PROGRAM UR5_robot
VAR
//banderas



i : BOOL := FALSE;
i2 : BOOL := FALSE;

vi_get_img : BOOL;
vi_img_ok: BOOL;

cx : REAL;
cy : REAL;
giro : REAL;
centro_ok : BOOL;
motor_pos_ok : BOOL;


// variables cabezal
giro_cabezal_dere : REAL;

vi_img_cabezal_dere_ok : BOOL;
vi_img_cabezal_dere_proc_ok : BOOL;
vi_get_img_cabezal_dere : BOOL;
vi_get_img_tuerca : BOOL;
giro_desartonillado : REAL;
cal_vueltas : REAL;
giro_aux_int : DINT;
giro_aux_float : REAL;

Atornillar: INT;
END_VAR

VAR_INPUT	
iniciar: BOOL := FALSE;
END_VAR

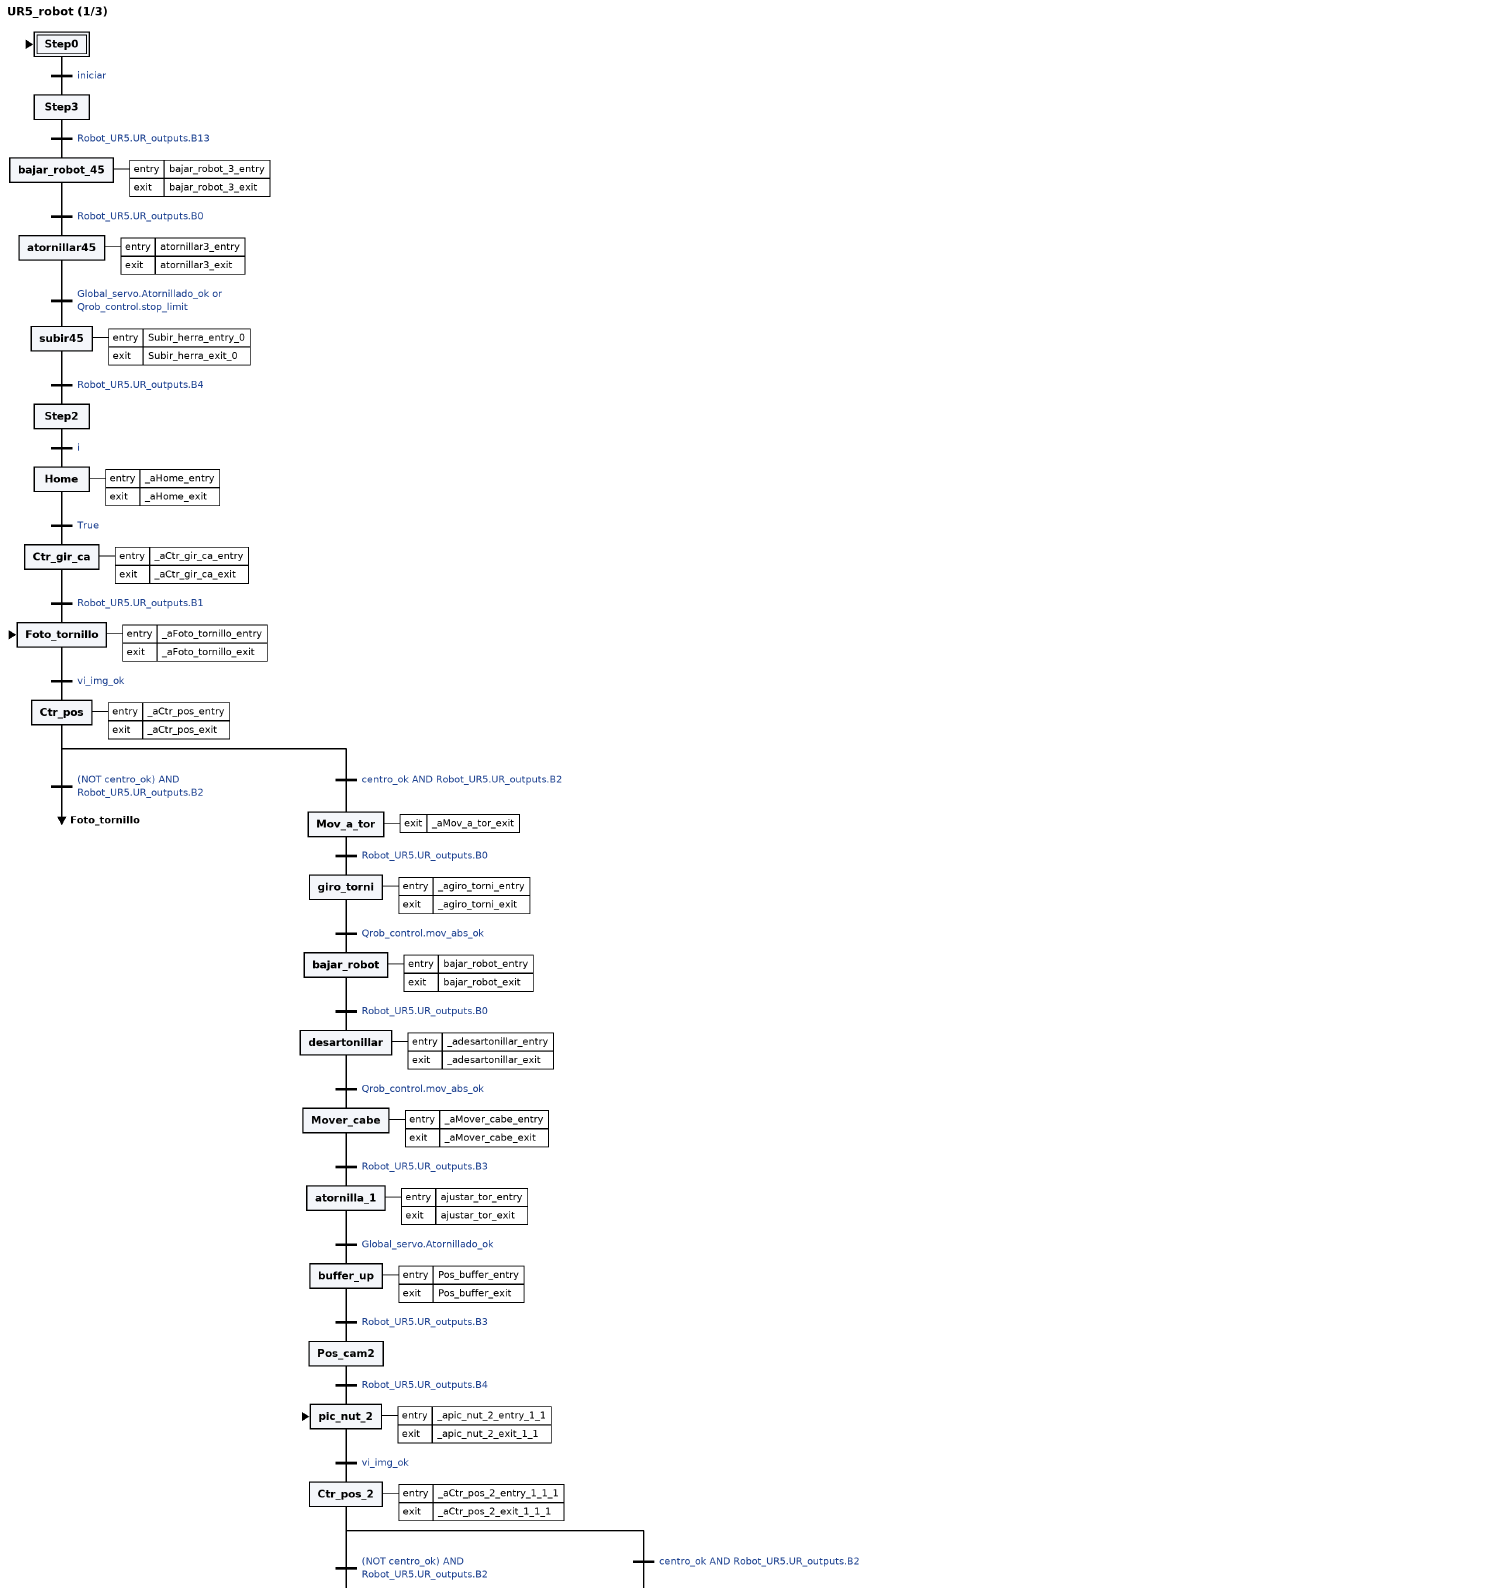
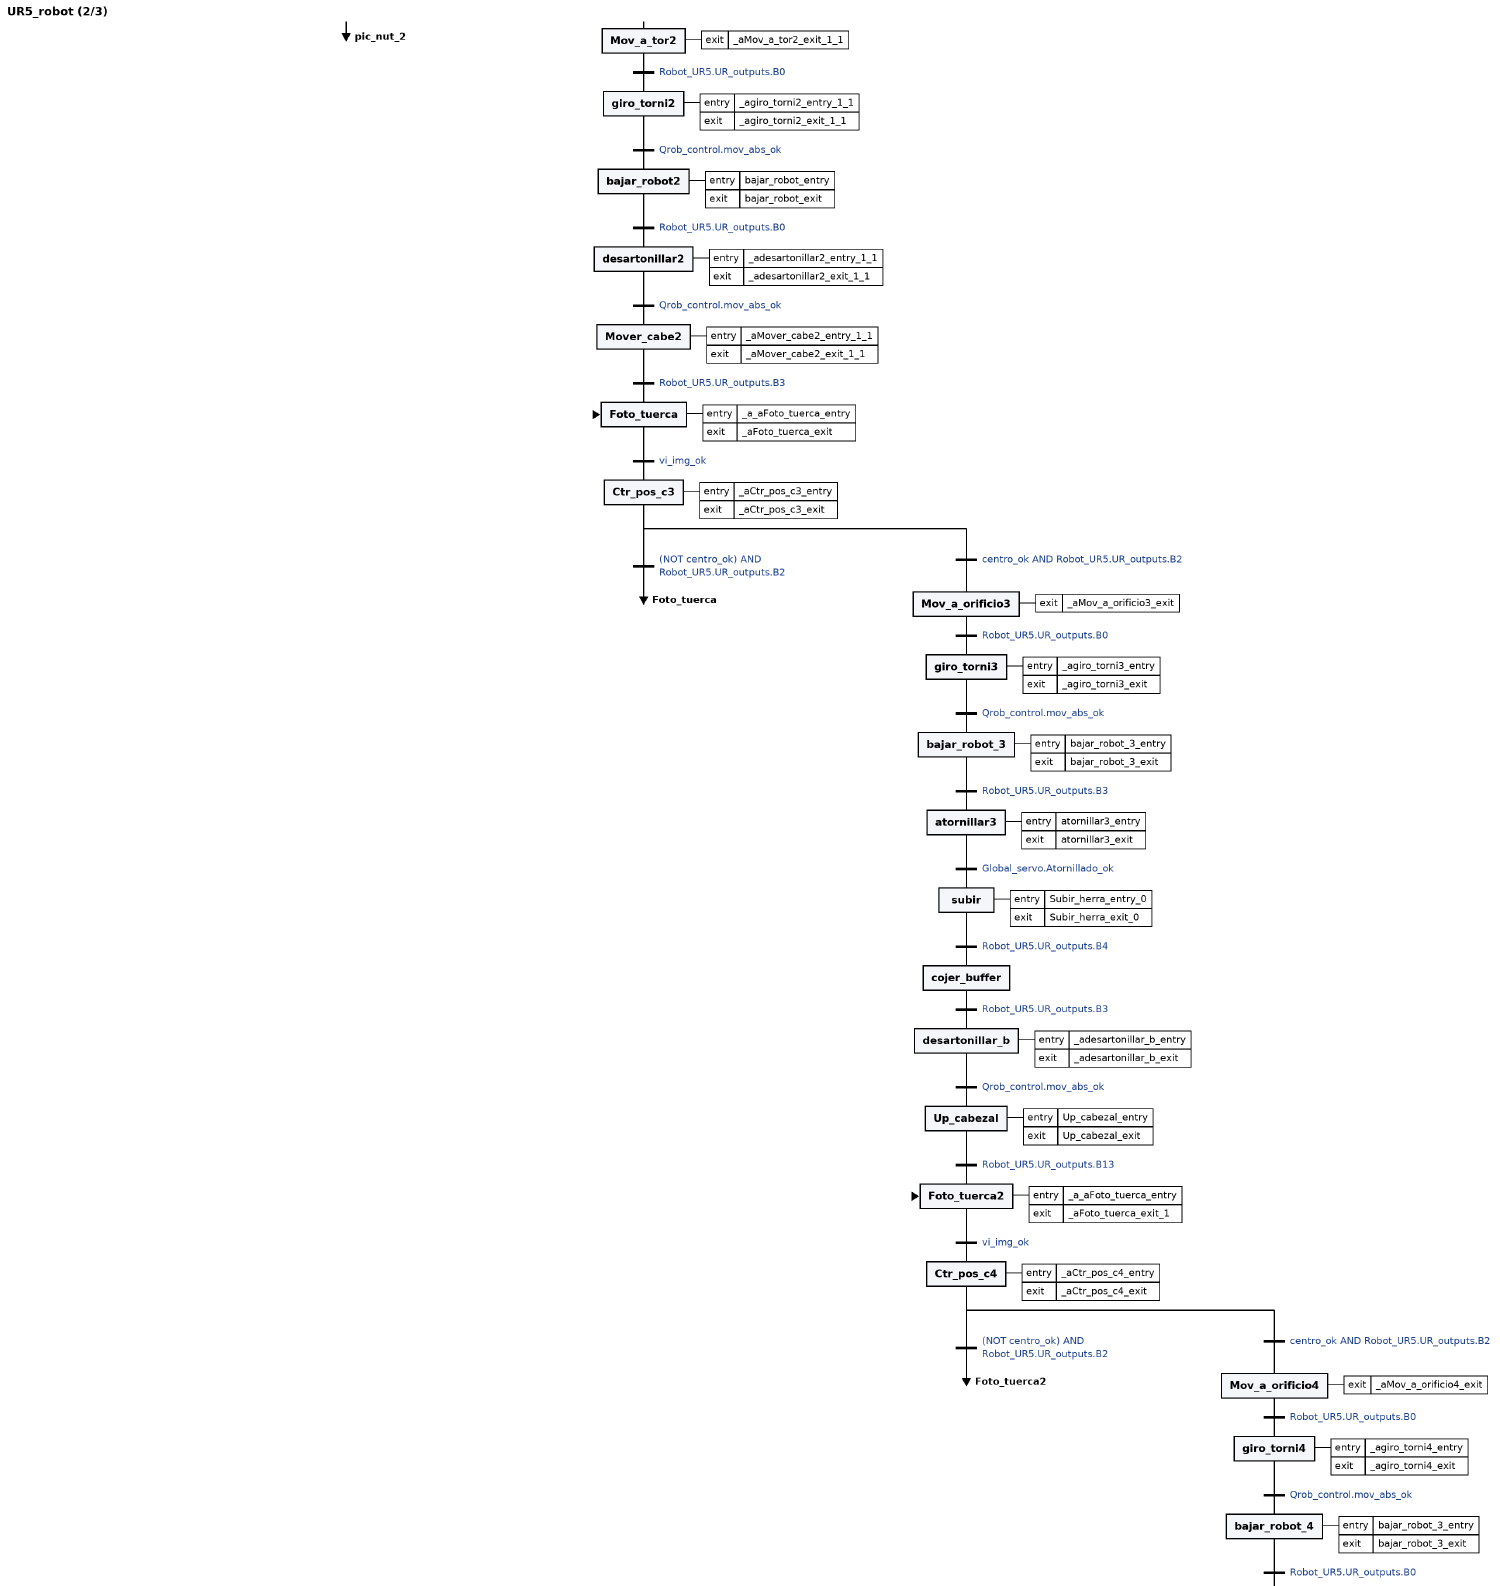
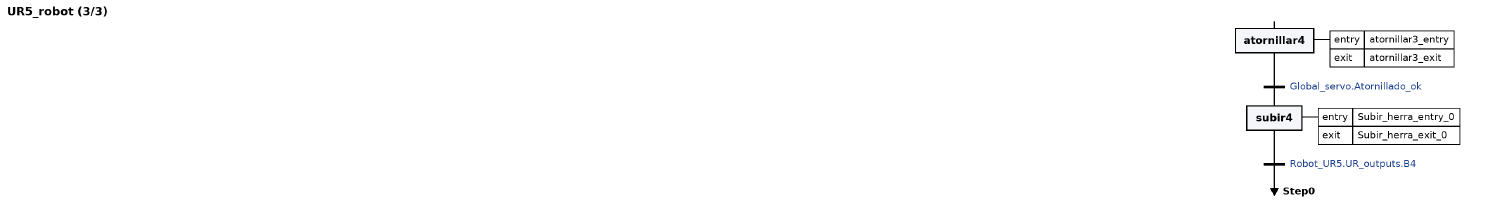
INITIAL_STEP Step0:
END_STEP
TRANSITION FROM Step0 TO Step3
    := iniciar;
END_TRANSITION
// macro Macro0 begins
STEP Step3:
END_STEP
TRANSITION FROM Step3 TO bajar_robot_45
    := Robot_UR5.UR_outputs.B13;
END_TRANSITION
STEP bajar_robot_45:
    bajar_robot_3_entry(P1);  // entry action
    bajar_robot_3_exit(P0);  // exit action
END_STEP
TRANSITION FROM bajar_robot_45 TO atornillar45
    := Robot_UR5.UR_outputs.B0;
END_TRANSITION
STEP atornillar45:
    atornillar3_entry(P1);  // entry action
    atornillar3_exit(P0);  // exit action
END_STEP
TRANSITION FROM atornillar45 TO subir45
    := Global_servo.Atornillado_ok or Qrob_control.stop_limit;
END_TRANSITION
STEP subir45:
    Subir_herra_entry_0(P1);  // entry action
    Subir_herra_exit_0(P0);  // exit action
END_STEP
TRANSITION FROM subir45 TO Step2
    := Robot_UR5.UR_outputs.B4;
END_TRANSITION
STEP Step2:
END_STEP
TRANSITION FROM Step2 TO Home
    := i;
END_TRANSITION
STEP Home:
    _aHome_entry(P1);  // entry action
    _aHome_exit(P0);  // exit action
END_STEP
TRANSITION FROM Home TO Ctr_gir_ca
    := True;
END_TRANSITION
STEP Ctr_gir_ca:
    _aCtr_gir_ca_entry(P1);  // entry action
    _aCtr_gir_ca_exit(P0);  // exit action
END_STEP
TRANSITION FROM Ctr_gir_ca TO Foto_tornillo
    := Robot_UR5.UR_outputs.B1;
END_TRANSITION
STEP Foto_tornillo:
    _aFoto_tornillo_entry(P1);  // entry action
    _aFoto_tornillo_exit(P0);  // exit action
END_STEP
TRANSITION FROM Foto_tornillo TO Ctr_pos
    := vi_img_ok;
END_TRANSITION
STEP Ctr_pos:
    _aCtr_pos_entry(P1);  // entry action
    _aCtr_pos_exit(P0);  // exit action
END_STEP
TRANSITION FROM Ctr_pos TO Foto_tornillo
    := (NOT centro_ok) AND Robot_UR5.UR_outputs.B2;
END_TRANSITION
TRANSITION FROM Ctr_pos TO Mov_a_tor
    := centro_ok AND Robot_UR5.UR_outputs.B2;
END_TRANSITION
STEP Mov_a_tor:
    _aMov_a_tor_exit(P0);  // exit action
END_STEP
TRANSITION FROM Mov_a_tor TO giro_torni
    := Robot_UR5.UR_outputs.B0;
END_TRANSITION
STEP giro_torni:
    _agiro_torni_entry(P1);  // entry action
    _agiro_torni_exit(P0);  // exit action
END_STEP
TRANSITION FROM giro_torni TO bajar_robot
    := Qrob_control.mov_abs_ok;
END_TRANSITION
STEP bajar_robot:
    bajar_robot_entry(P1);  // entry action
    bajar_robot_exit(P0);  // exit action
END_STEP
TRANSITION FROM bajar_robot TO desartonillar
    := Robot_UR5.UR_outputs.B0;
END_TRANSITION
STEP desartonillar:
    _adesartonillar_entry(P1);  // entry action
    _adesartonillar_exit(P0);  // exit action
END_STEP
TRANSITION FROM desartonillar TO Mover_cabe
    := Qrob_control.mov_abs_ok;
END_TRANSITION
STEP Mover_cabe:
    _aMover_cabe_entry(P1);  // entry action
    _aMover_cabe_exit(P0);  // exit action
END_STEP
TRANSITION FROM Mover_cabe TO atornilla_1
    := Robot_UR5.UR_outputs.B3;
END_TRANSITION
STEP atornilla_1:
    ajustar_tor_entry(P1);  // entry action
    ajustar_tor_exit(P0);  // exit action
END_STEP
TRANSITION FROM atornilla_1 TO buffer_up
    := Global_servo.Atornillado_ok;
END_TRANSITION
STEP buffer_up:
    Pos_buffer_entry(P1);  // entry action
    Pos_buffer_exit(P0);  // exit action
END_STEP
TRANSITION FROM buffer_up TO Pos_cam2
    := Robot_UR5.UR_outputs.B3;
END_TRANSITION
STEP Pos_cam2:
END_STEP
TRANSITION FROM Pos_cam2 TO pic_nut_2
    := Robot_UR5.UR_outputs.B4;
END_TRANSITION
STEP pic_nut_2:
    _apic_nut_2_entry_1_1(P1);  // entry action
    _apic_nut_2_exit_1_1(P0);  // exit action
END_STEP
TRANSITION FROM pic_nut_2 TO Ctr_pos_2
    := vi_img_ok;
END_TRANSITION
STEP Ctr_pos_2:
    _aCtr_pos_2_entry_1_1_1(P1);  // entry action
    _aCtr_pos_2_exit_1_1_1(P0);  // exit action
END_STEP
TRANSITION FROM Ctr_pos_2 TO pic_nut_2
    := (NOT centro_ok) AND Robot_UR5.UR_outputs.B2;
END_TRANSITION
TRANSITION FROM Ctr_pos_2 TO Mov_a_tor2
    := centro_ok AND Robot_UR5.UR_outputs.B2;
END_TRANSITION
STEP Mov_a_tor2:
    _aMov_a_tor2_exit_1_1(P0);  // exit action
END_STEP
TRANSITION FROM Mov_a_tor2 TO giro_torni2
    := Robot_UR5.UR_outputs.B0;
END_TRANSITION
STEP giro_torni2:
    _agiro_torni2_entry_1_1(P1);  // entry action
    _agiro_torni2_exit_1_1(P0);  // exit action
END_STEP
TRANSITION FROM giro_torni2 TO bajar_robot2
    := Qrob_control.mov_abs_ok;
END_TRANSITION
STEP bajar_robot2:
    bajar_robot_entry(P1);  // entry action
    bajar_robot_exit(P0);  // exit action
END_STEP
TRANSITION FROM bajar_robot2 TO desartonillar2
    := Robot_UR5.UR_outputs.B0;
END_TRANSITION
STEP desartonillar2:
    _adesartonillar2_entry_1_1(P1);  // entry action
    _adesartonillar2_exit_1_1(P0);  // exit action
END_STEP
TRANSITION FROM desartonillar2 TO Mover_cabe2
    := Qrob_control.mov_abs_ok;
END_TRANSITION
STEP Mover_cabe2:
    _aMover_cabe2_entry_1_1(P1);  // entry action
    _aMover_cabe2_exit_1_1(P0);  // exit action
END_STEP
TRANSITION FROM Mover_cabe2 TO Foto_tuerca
    := Robot_UR5.UR_outputs.B3;
END_TRANSITION
STEP Foto_tuerca:
    _a_aFoto_tuerca_entry(P1);  // entry action
    _aFoto_tuerca_exit(P0);  // exit action
END_STEP
TRANSITION FROM Foto_tuerca TO Ctr_pos_c3
    := vi_img_ok;
END_TRANSITION
STEP Ctr_pos_c3:
    _aCtr_pos_c3_entry(P1);  // entry action
    _aCtr_pos_c3_exit(P0);  // exit action
END_STEP
TRANSITION FROM Ctr_pos_c3 TO Foto_tuerca
    := (NOT centro_ok) AND Robot_UR5.UR_outputs.B2;
END_TRANSITION
TRANSITION FROM Ctr_pos_c3 TO Mov_a_orificio3
    := centro_ok AND Robot_UR5.UR_outputs.B2;
END_TRANSITION
STEP Mov_a_orificio3:
    _aMov_a_orificio3_exit(P0);  // exit action
END_STEP
TRANSITION FROM Mov_a_orificio3 TO giro_torni3
    := Robot_UR5.UR_outputs.B0;
END_TRANSITION
STEP giro_torni3:
    _agiro_torni3_entry(P1);  // entry action
    _agiro_torni3_exit(P0);  // exit action
END_STEP
TRANSITION FROM giro_torni3 TO bajar_robot_3
    := Qrob_control.mov_abs_ok;
END_TRANSITION
STEP bajar_robot_3:
    bajar_robot_3_entry(P1);  // entry action
    bajar_robot_3_exit(P0);  // exit action
END_STEP
TRANSITION FROM bajar_robot_3 TO atornillar3
    := Robot_UR5.UR_outputs.B3;
END_TRANSITION
STEP atornillar3:
    atornillar3_entry(P1);  // entry action
    atornillar3_exit(P0);  // exit action
END_STEP
TRANSITION FROM atornillar3 TO subir
    := Global_servo.Atornillado_ok;
END_TRANSITION
STEP subir:
    Subir_herra_entry_0(P1);  // entry action
    Subir_herra_exit_0(P0);  // exit action
END_STEP
TRANSITION FROM subir TO cojer_buffer
    := Robot_UR5.UR_outputs.B4;
END_TRANSITION
STEP cojer_buffer:
END_STEP
TRANSITION FROM cojer_buffer TO desartonillar_b
    := Robot_UR5.UR_outputs.B3;
END_TRANSITION
STEP desartonillar_b:
    _adesartonillar_b_entry(P1);  // entry action
    _adesartonillar_b_exit(P0);  // exit action
END_STEP
TRANSITION FROM desartonillar_b TO Up_cabezal
    := Qrob_control.mov_abs_ok;
END_TRANSITION
STEP Up_cabezal:
    Up_cabezal_entry(P1);  // entry action
    Up_cabezal_exit(P0);  // exit action
END_STEP
TRANSITION FROM Up_cabezal TO Foto_tuerca2
    := Robot_UR5.UR_outputs.B13;
END_TRANSITION
STEP Foto_tuerca2:
    _a_aFoto_tuerca_entry(P1);  // entry action
    _aFoto_tuerca_exit_1(P0);  // exit action
END_STEP
TRANSITION FROM Foto_tuerca2 TO Ctr_pos_c4
    := vi_img_ok;
END_TRANSITION
STEP Ctr_pos_c4:
    _aCtr_pos_c4_entry(P1);  // entry action
    _aCtr_pos_c4_exit(P0);  // exit action
END_STEP
TRANSITION FROM Ctr_pos_c4 TO Foto_tuerca2
    := (NOT centro_ok) AND Robot_UR5.UR_outputs.B2;
END_TRANSITION
TRANSITION FROM Ctr_pos_c4 TO Mov_a_orificio4
    := centro_ok AND Robot_UR5.UR_outputs.B2;
END_TRANSITION
STEP Mov_a_orificio4:
    _aMov_a_orificio4_exit(P0);  // exit action
END_STEP
TRANSITION FROM Mov_a_orificio4 TO giro_torni4
    := Robot_UR5.UR_outputs.B0;
END_TRANSITION
STEP giro_torni4:
    _agiro_torni4_entry(P1);  // entry action
    _agiro_torni4_exit(P0);  // exit action
END_STEP
TRANSITION FROM giro_torni4 TO bajar_robot_4
    := Qrob_control.mov_abs_ok;
END_TRANSITION
STEP bajar_robot_4:
    bajar_robot_3_entry(P1);  // entry action
    bajar_robot_3_exit(P0);  // exit action
END_STEP
TRANSITION FROM bajar_robot_4 TO atornillar4
    := Robot_UR5.UR_outputs.B0;
END_TRANSITION
STEP atornillar4:
    atornillar3_entry(P1);  // entry action
    atornillar3_exit(P0);  // exit action
END_STEP
TRANSITION FROM atornillar4 TO subir4
    := Global_servo.Atornillado_ok;
END_TRANSITION
STEP subir4:
    Subir_herra_entry_0(P1);  // entry action
    Subir_herra_exit_0(P0);  // exit action
END_STEP
TRANSITION FROM subir4 TO Step0
    := Robot_UR5.UR_outputs.B4;
END_TRANSITION

ACTION _a_aFoto_tuerca_entry:


vi_get_img_tuerca := True;
END_ACTION

ACTION _aCtr_gir_ca_entry:
Robot_UR5.UR_inputs.Floats.FLOAT3 := flip_real(data_to_robot.head_roll_right);
Robot_UR5.UR_inputs.Floats.FLOAT4 := flip_real(data_to_robot.head_roll_left);
Robot_UR5.UR_inputs.Bits.B0 := TRUE;
END_ACTION

ACTION _aCtr_gir_ca_exit:
Robot_UR5.UR_inputs.Bits.B0 := False;
END_ACTION

ACTION _aCtr_pos_2_entry_1_1_1:
vi_img_ok := FALSE;

Robot_UR5.UR_inputs.Floats.FLOAT0 := flip_real(cx);
Robot_UR5.UR_inputs.Floats.FLOAT1 := flip_real(cy);
Robot_UR5.UR_inputs.Floats.FLOAT2 := flip_real(giro);


IF ( ABS(cx) < 1) AND ( ABS(cy) < 1) THEN 
Robot_UR5.UR_inputs.Bits.B3 := TRUE;
centro_ok := TRUE;
ELSE 
Robot_UR5.UR_inputs.Bits.B3 := FALSE;
centro_ok := FALSE;	
END_IF

Robot_UR5.UR_inputs.Bits.B2 := TRUE;
END_ACTION

ACTION _aCtr_pos_2_exit_1_1_1:
Robot_UR5.UR_inputs.Bits.B2 := False;
END_ACTION

ACTION _aCtr_pos_c3_entry:
vi_img_ok := FALSE;

Robot_UR5.UR_inputs.Floats.FLOAT0 := flip_real(cx);
Robot_UR5.UR_inputs.Floats.FLOAT1 := flip_real(cy);



IF ( ABS(cx) < 0.5) AND ( ABS(cy) < 0.5) THEN 
Robot_UR5.UR_inputs.Bits.B3 := TRUE;
centro_ok := TRUE;
ELSE 
Robot_UR5.UR_inputs.Bits.B3 := FALSE;
centro_ok := FALSE;	
END_IF

Robot_UR5.UR_inputs.Bits.B2 := TRUE;
END_ACTION

ACTION _aCtr_pos_c3_exit:
Robot_UR5.UR_inputs.Bits.B2 := False;
END_ACTION

ACTION _aCtr_pos_c4_entry:
vi_img_ok := FALSE;

Robot_UR5.UR_inputs.Floats.FLOAT0 := flip_real(cx);
Robot_UR5.UR_inputs.Floats.FLOAT1 := flip_real(cy);



IF ( ABS(cx) < 0.5) AND ( ABS(cy) < 0.5) THEN 
Robot_UR5.UR_inputs.Bits.B3 := TRUE;
centro_ok := TRUE;
ELSE 
Robot_UR5.UR_inputs.Bits.B3 := FALSE;
centro_ok := FALSE;	
END_IF

Robot_UR5.UR_inputs.Bits.B2 := TRUE;
END_ACTION

ACTION _aCtr_pos_c4_exit:
Robot_UR5.UR_inputs.Bits.B2 := False;
END_ACTION

ACTION _aCtr_pos_entry:
vi_img_ok := FALSE;

Robot_UR5.UR_inputs.Floats.FLOAT0 := flip_real(cx);
Robot_UR5.UR_inputs.Floats.FLOAT1 := flip_real(cy);
Robot_UR5.UR_inputs.Floats.FLOAT2 := flip_real(giro);


IF ( ABS(cx) < 1) AND ( ABS(cy) < 1) THEN 
Robot_UR5.UR_inputs.Bits.B3 := TRUE;
centro_ok := TRUE;
ELSE 
Robot_UR5.UR_inputs.Bits.B3 := FALSE;
centro_ok := FALSE;	
END_IF

Robot_UR5.UR_inputs.Bits.B2 := TRUE;
END_ACTION

ACTION _aCtr_pos_exit:
Robot_UR5.UR_inputs.Bits.B2 := False;
END_ACTION

ACTION _adesartonillar_b_entry:




giro_desartonillado :=  (-24*360) + Qrob_control.actual_position;
Qrob_control.pos_mover_abs := giro_desartonillado;
Qrob_control.velocidad := 150;


Qrob_control.mover_abs := TRUE;
END_ACTION

ACTION _adesartonillar_b_exit:
Qrob_control.mover_abs := FALSE;
END_ACTION

ACTION _adesartonillar_entry:




giro_desartonillado := giro -(15*360);
//giro_desartonillado := giro -2160;
Qrob_control.pos_mover_abs := giro_desartonillado;
Qrob_control.velocidad := 150;


Qrob_control.mover_abs := TRUE;
END_ACTION

ACTION _adesartonillar_exit:
Qrob_control.mover_abs := FALSE;
END_ACTION

ACTION _adesartonillar2_entry_1_1:





giro_desartonillado := giro -(15*360);
//giro_desartonillado := giro -2160;
Qrob_control.pos_mover_abs := giro_desartonillado;
Qrob_control.velocidad := 150;


Qrob_control.mover_abs := TRUE;
END_ACTION

ACTION _adesartonillar2_exit_1_1:
Qrob_control.mover_abs := FALSE;
END_ACTION

ACTION _aFoto_tornillo_entry:
vi_get_img := True;
END_ACTION

ACTION _aFoto_tornillo_entry_1:
vi_get_img := True;
END_ACTION

ACTION _aFoto_tornillo_exit:
vi_get_img := False;
END_ACTION

ACTION _aFoto_tuerca_exit:

vi_get_img_tuerca := False;
END_ACTION

ACTION _aFoto_tuerca_exit_1:

vi_get_img_tuerca := False;
END_ACTION

ACTION _agiro_torni_entry:
//POU.detener := TRUE;
//Pou.detener := FALSE;


//home qrob while angle
giro_aux_int := ABS(TRUNC(Qrob_control.actual_position/360));
giro_aux_float := ABS( - (Qrob_control.actual_position/360));
giro_aux_float := -1*(giro_aux_float*360);






Qrob_control.velocidad := 50;
//Qrob_control.pos_mover_abs := giro;
Qrob_control.pos_mover_abs := (Qrob_control.actual_position + giro_aux_float) + giro;
Qrob_control.mover_abs := TRUE;
END_ACTION

ACTION _agiro_torni_exit:
Qrob_control.mover_abs := FALSE;
END_ACTION

ACTION _agiro_torni2_entry_1_1:
//POU.detener := TRUE;
//Pou.detener := FALSE;


//home qrob while angle
giro_aux_int := ABS(TRUNC(Qrob_control.actual_position/360));
giro_aux_float := ABS(giro_aux_int- (Qrob_control.actual_position/360));
giro_aux_float := -1*(giro_aux_float*360);






Qrob_control.velocidad := 50;
//Qrob_control.pos_mover_abs := giro;
Qrob_control.pos_mover_abs := (Qrob_control.actual_position + giro_aux_float) + giro;
giro := Qrob_control.pos_mover_abs;
Qrob_control.mover_abs := TRUE;
END_ACTION

ACTION _agiro_torni2_exit_1_1:
Qrob_control.mover_abs := FALSE;
END_ACTION

ACTION _agiro_torni3_entry:
//POU.detener := TRUE;
//Pou.detener := FALSE;


giro_aux_int := TRUNC(Qrob_control.actual_position/360);

giro_aux_float := ABS(giro_aux_int- (Qrob_control.actual_position/360));
giro_aux_float := -1*(giro_aux_float*360);

Qrob_control.velocidad := 100;
Qrob_control.pos_mover_abs := Qrob_control.actual_position + giro_aux_float;
Qrob_control.mover_abs := TRUE;
END_ACTION

ACTION _agiro_torni3_exit:
Qrob_control.mover_abs := FALSE;
END_ACTION

ACTION _agiro_torni4_entry:
//POU.detener := TRUE;
//Pou.detener := FALSE;

//Qrob_control.velocidad := 100;
//Qrob_control.pos_mover_abs := 0;
//Qrob_control.mover_abs := TRUE;


giro_aux_int := TRUNC(Qrob_control.actual_position/360);

giro_aux_float := ABS(giro_aux_int- (Qrob_control.actual_position/360));
giro_aux_float := -1*(giro_aux_float*360);

Qrob_control.velocidad := 100;
Qrob_control.pos_mover_abs := Qrob_control.actual_position + giro_aux_float;
Qrob_control.mover_abs := TRUE;
END_ACTION

ACTION _agiro_torni4_exit:
Qrob_control.mover_abs := FALSE;
END_ACTION

ACTION _aHome_entry:
i := FALSE;
Robot_UR5.UR_inputs.Bits.B0 := TRUE;
//POU.EnableAxis1 := True;
giro :=0;
//Qrob_control.ajustar_tornillo := FALSE;
//Qrob_control.pos_mover_abs := 0;
//Qrob_control.velocidad := 100;


//Qrob_control.mover_abs := TRUE;
END_ACTION

ACTION _aHome_exit:
Robot_UR5.UR_inputs.Bits.B0 := FALSE;
iniciar := FALSE;
Qrob_control.mover_abs := False;
END_ACTION

ACTION _aMov_a_orificio3_exit:
Robot_UR5.UR_inputs.Bits.B2 := FALSE;
END_ACTION

ACTION _aMov_a_orificio4_exit:
Robot_UR5.UR_inputs.Bits.B2 := FALSE;
END_ACTION

ACTION _aMov_a_tor_exit:
Robot_UR5.UR_inputs.Bits.B2 := FALSE;
END_ACTION

ACTION _aMov_a_tor2_exit_1_1:
Robot_UR5.UR_inputs.Bits.B2 := FALSE;
END_ACTION

ACTION _aMover_cabe_entry:
Robot_UR5.UR_inputs.Bits.B5 := True;
END_ACTION

ACTION _aMover_cabe_exit:
Robot_UR5.UR_inputs.Bits.B5 := False;
END_ACTION

ACTION _aMover_cabe2_entry_1_1:
Robot_UR5.UR_inputs.Bits.B5 := True;
END_ACTION

ACTION _aMover_cabe2_exit_1_1:
Robot_UR5.UR_inputs.Bits.B5 := False;
END_ACTION

ACTION _apic_nut_2_entry_1_1:
vi_get_img := True;
END_ACTION

ACTION _apic_nut_2_exit_1_1:
vi_get_img := False;
END_ACTION

ACTION ajustar_tor_entry:


//Atornillado_funcion(Iniciar:= TRUE, Corriente := 60, vueltas := 8, giro_alivio := 3);

Atornillar_CS.UR5.Corriente := 10;
Atornillar_CS.UR5.Vueltas := 21;
Atornillar_CS.UR5.Iniciar := TRUE;
END_ACTION

ACTION ajustar_tor_exit:
Global_servo.Atornillado_ok := FALSE;
Atornillar_CS.UR5.Iniciar := FALSE;
END_ACTION

ACTION atornillar_2_entry:

Atornillar_CS.UR5.Corriente :=100;
Atornillar_CS.UR5.Vueltas := 4;
Atornillar_CS.UR5.Iniciar := True;
END_ACTION

ACTION atornillar_2_exit:
Global_servo.Atornillado_ok := FALSE;
Atornillar_CS.UR5.Iniciar := False;
END_ACTION

ACTION atornillar3_entry:

//Atornillado_funcion(Iniciar:= TRUE, Corriente := 60, vueltas := 8, giro_alivio := 3);

//Atornillar_CS.UR5.Corriente := 75;
//Atornillar_CS.UR5.Vueltas := 13;
//Atornillar_CS.UR5.Iniciar := TRUE;

Qrob_control.ajustar_tornillo := TRUE;
Qrob_control.limite_corriente := 150;
Qrob_control.mover_horario := TRUE;
END_ACTION

ACTION atornillar3_exit:
//Global_servo.Atornillado_ok := FALSE;
//Atornillar_CS.UR5.Iniciar := FALSE;



Qrob_control.ajustar_tornillo := FALSE;
Qrob_control.limite_corriente := 100;
Qrob_control.mover_horario := FALSE;
Qrob_control.detener := FALSE;
END_ACTION

ACTION bajar_robot_3_entry:

Robot_UR5.UR_inputs.Bits.B0 := TRUE;
END_ACTION

ACTION bajar_robot_3_exit:
Robot_UR5.UR_inputs.Bits.B0 := FALSE;
Robot_UR5.UR_inputs.Bits.B10 := False;
END_ACTION

ACTION bajar_robot_entry:
Robot_UR5.UR_inputs.Bits.B0 := TRUE;
END_ACTION

ACTION bajar_robot_exit:
Robot_UR5.UR_inputs.Bits.B0 := False;
END_ACTION

ACTION Cabe_separador_entry:
Robot_UR5.UR_inputs.Bits.B5 := TRUE;
END_ACTION

ACTION Cabe_separador_exit:
Robot_UR5.UR_inputs.Bits.B5 := False;
END_ACTION

ACTION Pos_buffer_entry:

Robot_UR5.UR_inputs.Bits.B7 := TRUE;
END_ACTION

ACTION Pos_buffer_exit:

Robot_UR5.UR_inputs.Bits.B7 := False;
END_ACTION

ACTION Step1_entry:
Robot_UR5.UR_inputs.Bits.B7 := TRUE;
END_ACTION

ACTION Step1_exit:
Robot_UR5.UR_inputs.Bits.B7 := False;
END_ACTION

ACTION Subir_herra_entry:
Robot_UR5.UR_inputs.Bits.B7 := TRUE;
Qrob_control.detener := TRUE;
Qrob_control.detener := FALSE;


Robot_UR5.UR_inputs.Bits.B7 := TRUE;
Qrob_control.pos_mover_abs := Qrob_control.actual_position -10;




Qrob_control.velocidad := 1;
Qrob_control.mover_abs := TRUE;
END_ACTION

ACTION Subir_herra_entry_0:
Robot_UR5.UR_inputs.Bits.B5 := TRUE;
Robot_UR3.UR_outputs.B6 := False;
END_ACTION

ACTION Subir_herra_exit:
Robot_UR5.UR_inputs.Bits.B7 := FALSE;
Qrob_control.mover_abs := FALSE;
END_ACTION

ACTION Subir_herra_exit_0:
Robot_UR5.UR_inputs.Bits.B5 := FALSE;
Robot_UR3.UR_outputs.B6 := True;
END_ACTION

ACTION Up_cabezal_entry:
Robot_UR5.UR_inputs.Bits.B8 := TRUE;
END_ACTION

ACTION Up_cabezal_exit:
Robot_UR5.UR_inputs.Bits.B8 := False;
END_ACTION

END_PROGRAM

(* stored: Version 1.1.0.1, ProductVersion 3.1.4024.4
   POU UR5_robot: Id {1c1a3202-8aac-4f16-ba80-1c87a68e2de2}, SpecialFunc None
   Action _a_aFoto_tuerca_entry: Id {ee0ad9a1-c258-412a-913f-33db82c95a06}
   Action _aCtr_gir_ca_entry: Id {6badef7f-2aff-4f85-b5da-0017cf53224d}
   Action _aCtr_gir_ca_exit: Id {925f140e-d69c-4f0a-885e-621ee159b154}
   Action _aCtr_pos_2_entry_1_1_1: Id {59038164-db62-4fd6-abfa-808281c1dfd4}
   Action _aCtr_pos_2_exit_1_1_1: Id {c2b52dd7-be97-4c93-9697-de96d05d47fe}
   Action _aCtr_pos_c3_entry: Id {e1ccd9dd-d58a-49f1-ad40-a7a2e78cbf69}
   Action _aCtr_pos_c3_exit: Id {d51d8321-e5fc-4626-b50a-1d098057cc3d}
   Action _aCtr_pos_c4_entry: Id {c3ee579b-75cb-4396-af88-28df648d5d65}
   Action _aCtr_pos_c4_exit: Id {0d3f0d94-2264-4971-a4b8-5d9de697d443}
   Action _aCtr_pos_entry: Id {6e7eba6f-6db5-47b1-b14b-435b37d220bf}
   Action _aCtr_pos_exit: Id {afdf3cfc-7faf-407c-9460-b385a465837a}
   Action _adesartonillar_b_entry: Id {5aaa2efd-ed00-4002-9625-27976925f455}
   Action _adesartonillar_b_exit: Id {68d9b5ed-e446-49ec-ade2-e68bd4ada3d9}
   Action _adesartonillar_entry: Id {2f4a0c66-5f49-4a1e-89b3-fd3390dc547f}
   Action _adesartonillar_exit: Id {066017be-1043-4afd-9913-fb9e38539fb5}
   Action _adesartonillar2_entry_1_1: Id {020ac4a9-7ecd-493c-83da-de05e4d6735e}
   Action _adesartonillar2_exit_1_1: Id {ec708201-346d-41df-8644-5b24542a2676}
   Action _aFoto_tornillo_entry: Id {284889eb-2191-4c5e-bdfc-12becc321b36}
   Action _aFoto_tornillo_entry_1: Id {8a63648a-27a6-4461-9145-c57f8136e669}
   Action _aFoto_tornillo_exit: Id {f05c2629-852e-4e18-a2e7-0c2df1e2f22b}
   Action _aFoto_tuerca_exit: Id {8661d695-e134-4700-9ffe-202f26f2cec0}
   Action _aFoto_tuerca_exit_1: Id {b31a8ca8-c5c4-4fd4-80b9-99f0139693e7}
   Action _agiro_torni_entry: Id {95fb54c7-1fd8-41c6-a901-4180861c4d03}
   Action _agiro_torni_exit: Id {26a027b7-af17-4be1-91fc-c24be3f80b36}
   Action _agiro_torni2_entry_1_1: Id {b0c15ecd-2bb5-47bc-a974-1df607ee723c}
   Action _agiro_torni2_exit_1_1: Id {adf7b5c3-916b-478d-9248-8f18eb5b398c}
   Action _agiro_torni3_entry: Id {c519d598-d895-48ee-80df-d8a8542f81e5}
   Action _agiro_torni3_exit: Id {c5e90149-a683-4487-9fd1-c28933f6a75c}
   Action _agiro_torni4_entry: Id {82fee7b9-1ce7-4d1e-a28c-57be461b9e80}
   Action _agiro_torni4_exit: Id {304b5ded-44f6-488f-a2e6-b2ca8723e8e1}
   Action _aHome_entry: Id {d455378b-e6f2-4c4e-86e3-3eba108c6d09}
   Action _aHome_exit: Id {5321d8cf-929c-4243-8d4d-a3348397546c}
   Action _aMov_a_orificio3_exit: Id {4411de4c-f59b-4388-ac7f-5484da707aa8}
   Action _aMov_a_orificio4_exit: Id {de397a07-c9da-49ab-b7ea-5f2b0874167a}
   Action _aMov_a_tor_exit: Id {b3bc6c24-1bda-4ad7-95ba-1ab58ab559b2}
   Action _aMov_a_tor2_exit_1_1: Id {997279d3-cd92-4895-9445-68709b3e3269}
   Action _aMover_cabe_entry: Id {008cc0ab-8abb-415b-b328-71c5a120f70c}
   Action _aMover_cabe_exit: Id {59b99ff1-ca14-4ed0-bf72-a5dd234ae849}
   Action _aMover_cabe2_entry_1_1: Id {39b56a71-f556-4b9d-9cab-45b89a79b32c}
   Action _aMover_cabe2_exit_1_1: Id {911fb5b9-386d-4810-af20-9a8e136c35c0}
   Action _apic_nut_2_entry_1_1: Id {b3ea873c-f2c5-49f7-9870-6e1572adf631}
   Action _apic_nut_2_exit_1_1: Id {58c4fbcc-6395-4ffb-9ba0-ea5374886325}
   Action ajustar_tor_entry: Id {b9be4c25-1b93-4d76-b349-e25471b98da1}
   Action ajustar_tor_exit: Id {cc862e8c-0df4-431c-9b3c-32fdfe851778}
   Action atornillar_2_entry: Id {9bd55512-3c14-4b68-9b71-3b32f97a24e5}
   Action atornillar_2_exit: Id {6ac4439f-69fa-4a7d-9488-b3e8397d00c1}
   Action atornillar3_entry: Id {de8bc843-ef18-4615-82a1-2e44df9c638a}
   Action atornillar3_exit: Id {255d2952-0ad3-42f8-bdd7-c5f5f39f63ca}
   Action bajar_robot_3_entry: Id {d9d8038c-a269-41cc-8a3f-4470dab230ab}
   Action bajar_robot_3_exit: Id {642d9cb1-e355-4f37-9a7d-383f37e2909f}
   Action bajar_robot_entry: Id {e4c0dbf5-0e0a-4d6b-a7c9-dbf2ee518f98}
   Action bajar_robot_exit: Id {1dcb9c72-0ad6-40c1-9dc2-284a3f25cdad}
   Action Cabe_separador_entry: Id {cf3e6dd4-f088-49ae-9c10-01323c6b5ba6}
   Action Cabe_separador_exit: Id {99aede7a-a449-4b94-b479-7347f4a58801}
   Action Pos_buffer_entry: Id {0dc12635-c58b-419b-a4ba-a9f80d727d13}
   Action Pos_buffer_exit: Id {059b1db5-f51c-46c8-b768-ea3f2a35ab58}
   Action Step1_entry: Id {7965ab5f-94b8-414e-9c61-956e59652ea2}
   Action Step1_exit: Id {81f6eb1b-b6fd-4b7d-8616-b5d9cb705615}
   Action Subir_herra_entry: Id {f472e93e-fb4d-4977-ad48-84211f85e07f}
   Action Subir_herra_entry_0: Id {9fa17653-87d7-4c09-a3d7-1cf7ef23a6c8}
   Action Subir_herra_exit: Id {ac5eda4e-ca59-4ac4-a8d8-c5c6ae533909}
   Action Subir_herra_exit_0: Id {9242a96d-7824-4cb1-8c1f-ef8a61e130fc}
   Action Up_cabezal_entry: Id {2ee65113-8c81-4e63-9a58-b891b386eefd}
   Action Up_cabezal_exit: Id {5ec6b1f3-c3c7-4acf-af2d-bf8709a1579f} *)
